PROGRAM MAIN
VAR
	bTasterBlau 	: BOOL := TRUE; //bool
	uiZaehlerObjekt	: UINT := 23; //uint 16bit
	rTemp			: REAL := -3.34; //float 16bit
	(*
	Kommentar
	*)
	rAdditionResult : REAL;
END_VAR

IF bTasterBlau THEN
	uiZaehlerObjekt := uiZaehlerObjekt +1;
END_IF

rAdditionResult := F_AdditionFunction(4.3,3.4);

PRG_DoSomeMath();

END_PROGRAM

(* stored: Version 1.1.0.1, ProductVersion 3.1.4024.13
   POU MAIN: Id {e16cbd2e-88ff-4213-8f72-3fa553782b4d}, SpecialFunc None *)
